Yaskawa INFORM job: NETFTS_BIAS.JBI

/JOB
//NAME NETFTS_BIAS
///FOLDERNAME NETFTS_FORCETORQUESENSOR
//POS
///NPOS 0,0,0,0,0,0
//INST
///DATE 2021/10/18 12:49
///COMM Used By Ethernet FT Sensor Ext
///ATTR SC,RW
///GROUP1 RB1
///LVARS 1,0,0,0,0,0,0,0
NOP
SET LB000 B[80]
ADD LB000 1
VAL B[LB000] "1"
TIMER T=0.50
VAL B[LB000] "0"
END
